{attribute 'qualified_only'}
// ***********************************************************************************
//
// USI Mendrisio, Largo Bernasconi 2, CH-6850 Mendrisio
// ETH Zurich, Building HIF E26, Laura-Hezner-Weg 7, CH-8093 Zürich
//
// ***********************************************************************************
//
// PROJECT     :  Clay Printing Controller
// FUNCTION    :  README
// AUTHOR      :  WeiTing Chen
// EMAIL       :  chen@mesh.ch
// Copyright   :  USI FMAA Mendrisio(CH) 2025
//
// ***********************************************************************************

VAR_GLOBAL
(*
Set the IP with XXXXXXXX

File description
GVL(GVL : Global variables)
GVL_IO(GVL_IO : IO)
GVL_LAP(GVL_LAP : variables for control via laptop)

Data Type Prefix
ib = Input Bool   / ob = Output Bool
if = Input float  / of = Output float (REAL, LREAL)
in = Input numeric/ on = Output numeric
(INT, SINT, USINT, UNIT, DINT, UDINT, BYTE, WORD, DWORD, LWORD, XINT, UXINT, XWORD)
t = Time (TON)
s = String

Naming Shortcuts
CC1 = Concrete Controller
CP1 = Concrete Pump
PN = Profinet with Roboter

*)
END_VAR

(* stored: Version 1.1.0.1, ProductVersion 3.1.4024.15
   GVL README: Id {323cccd0-94c1-445f-830c-f2af6b81bf72} *)
